Universal Robots PolyScope program: TEST_SUB_106.urp

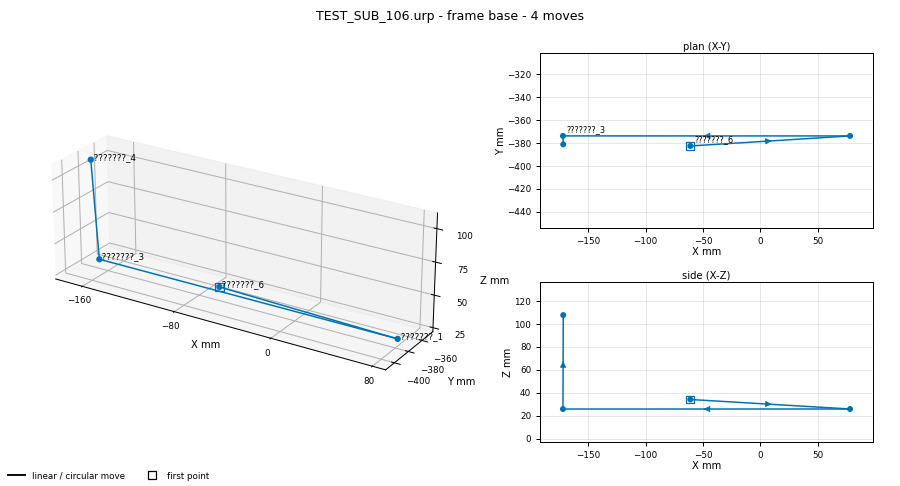
[picture p0: tool path of TEST_SUB_106.urp in frame base, 4 of 4 moves have a stored position in this frame; points joined in program order, loops and branches not executed]
Program TEST_SUB_106 (installation=GD directory=/programs/GD createdIn=5.13.0 lastSavedIn=5.13.0 robotSerialNumber=20205000017)
Calibrated DH parameters: a=[-0.000157, -0.56303, -0.236706, -0.000074, -0.000109, 0]; d=[0.181705, 47.632387, 369.599619, -417.058513, 0.119878, 0.115667]; alpha=[1.570881, -0.005074, -0.001247, 1.56886, -1.570997, 0]; deltaTheta=[0, -0.405485, 5.544791, 1.143886, -0.000009, -0.000001]
InitVariablesNode
Robot Program (runOnlyOnce=false)
  var_4 := p[0.0,0.0,0.0,CutOffPos[3],CutOffPos[4],CutOffPos[5]]
  var_5 := p[0.0,0.0,0.0,CutOffPos[3],CutOffPos[4],CutOffPos[5]]
  Script: CurrPos=get_actual_tool_flange_pose()
  CutOffPos := CurrPos
  var_1 := get_tcp_offset()
  var_2 := pose_trans(CutOffPos,var_1)
  MoveL speed 250 mm/s, acceleration 50 mm/s^2 (useActiveTCP=false) tcp=TCP_1; feature=Base
    SuppressedNode
      var_3 := get_tcp_offset()
    SuppressedNode
      Waypoint ウェイポイント_2: TCP in base x=-24.264 y=-372.872 z=25.863 mm, rx=-0.0592 ry=3.141 rz=-0.0002 rad; joints [-70.474, -66.693, -131.957, -71.332, 89.989, 17.477] deg; TCP offset x=0 y=80 z=420 mm, rx=0 ry=0 rz=0 rad
    SuppressedNode
      Wait Sleep waitTime=0.5
    Waypoint ウェイポイント_6: TCP in base x=-61.068 y=-382.464 z=34.138 mm, rx=0.7542 ry=-2.9409 rz=0.2397 rad; joints [-60.318, -53.474, -138.479, -70.758, 82.346, 0.532] deg
    Wait Sleep waitTime=0.5
  SuppressedNode
    Folder FREE_DRIVE
      Script: freedrive_mode()
      SetPayload (workpieceName=k2)
      Set NoAction tcp=ZERO
      Wait Sleep waitTime=1
      Script: end_freedrive_mode()
      Wait Condition expression=is_steady()
  SetPayload (workpieceName=k10)
  Set NoAction tcp=TCP_1
  Wait Sleep waitTime=0.5
  Folder CUTOFF_POSE
    CutOffPos := CurrPos
    var_6 := CutOffPos
    SuppressedNode
      CutOffPos := p[0.0,0.0,0.0,CutOffPos[3],CutOffPos[4],CutOffPos[5]]
    var_1 := get_tcp_offset()
    var_20 := pose_trans(pose_inv(CutOffPos),var_1)
    SuppressedNode
      CutOffPos := 
    var_4 := p[0.0,0.0,0.0,CutOffPos[3],CutOffPos[4],CutOffPos[5]]
    var_5 := p[0.0,0.0,0.0,0.0,0.0,CutOffPos[5]]
    CutOffPos := pose_trans(var_4,pose_inv(var_5))
    SuppressedNode
      CutOffPos := p[0.0,0.0,0.0,var_5[0],var_5[1],var_5[2]]
    var_20 := pose_trans(pose_inv(CutOffPos),var_1)
    var_21 := pose_trans(var_1,CutOffPos)
    var_2 := pose_trans(CutOffPos,var_1)
  Wait Condition expression=is_steady()
  SuppressedNode
    Script: CurrPos_p=get_actual_tcp_pose()
  SuppressedNode
    CircleMove (OrientationMode=UNCONSTRAINED)
  Script: set_tcp(var_2)
  SuppressedNode
    Folder TRANSFER
      Timer (action=Reset) variable(name=tm_relmove)
      Timer (action=Start) variable=tm_relmove
      ForceStartZ := CurrPos_p[2]
      Force Frame feature=Bucket; selection=[0, 0, 1, 0, 0, 0]; wrench=[0, 0, 40, 0, 0, 0]; limitsForce=[0.01, 0.01, 0.25, 0.174533, 0.174533, 0.174533]; limitsMotion=[0.1, 0.1, 0.1, 0.349066, 0.349066, 0.349066]
        Wait Condition expression=tm_relmove>GPII_TMCutOff or CurrPos_p[2]>ForceStartZ+RelMoveZ
      Timer (action=Stop) variable=tm_relmove
      If (WorkPosNo≟0)
        MoveL speed 60 mm/s, acceleration 15 mm/s^2 (useActiveTCP=false) tcp=ZERO; feature=Base
          PoseSub := pose_sub(CurrPos, pose_trans(g2GD_pos5, pose_inv(get_tcp_offset())))
          RZSub := r2d(PoseSub[5])
          If (norm(PoseSub[5])≥d2r(RZTh))
            Script: PoseSub[0]=0.0
            Script: PoseSub[1]=0.0
            Script: PoseSub[2]=0.0
            PoseAdd := pose_add(PoseSub, CurrPos)
            Waypoint Variable (Variable): variable=PoseAdd
        MoveL speed 250 mm/s, acceleration 50 mm/s^2 (useActiveTCP=false) tcp=TCP_1; feature=Base
          Waypoint Variable (Variable): variable(featureName=g2GD_pos5)
        MoveL speed 400 mm/s, acceleration 140 mm/s^2 (useActiveTCP=false) tcp=TCP_1; feature=Base
          SetPayload (workpieceName=k10)
          Waypoint Variable (Variable): variable(featureName=g2GD_pos4)
          Waypoint Variable (Variable): motionParameters(blendRadius=0.1); variable(featureName=g2GD_pos3)
          Waypoint Variable (Variable): motionParameters(jointSpeed=1.047198 jointAcceleration=1.396263 cartesianSpeed=0.4 cartesianAcceleration=0.07); variable(featureName=g2GD_pos2)
        MoveL speed 400 mm/s, acceleration 70 mm/s^2 (useActiveTCP=false) tcp=TCP_1; feature=Base
          SetPayload (workpieceName=k120)
          Waypoint Variable (Variable): motionParameters(blendRadius=0.05); variable(featureName=g2GD_pos1)
      ElseIf (WorkPosNo≟1)
        MoveL speed 60 mm/s, acceleration 15 mm/s^2 (useActiveTCP=false) tcp=ZERO; feature=Base
          PoseSub := pose_sub(CurrPos, pose_trans(g1GD_pos5, pose_inv(get_tcp_offset())))
          RZSub := r2d(PoseSub[5])
          If (norm(PoseSub[5])≥d2r(RZTh))
            Script: PoseSub[0]=0.0
            Script: PoseSub[1]=0.0
            Script: PoseSub[2]=0.0
            PoseAdd := pose_add(PoseSub, CurrPos)
            Waypoint Variable (Variable): variable=PoseAdd
        MoveL speed 250 mm/s, acceleration 50 mm/s^2 (useActiveTCP=false) tcp=TCP_1; feature=Base
          Waypoint Variable (Variable): variable(featureName=g1GD_pos5)
        MoveL speed 400 mm/s, acceleration 140 mm/s^2 (useActiveTCP=false) tcp=TCP_1; feature=Base
          SetPayload (workpieceName=k10)
          Waypoint Variable (Variable): variable(featureName=g1GD_pos3)
          Waypoint Variable (Variable): variable(featureName=g1GD_pos2)
        MoveL speed 400 mm/s, acceleration 140 mm/s^2 (useActiveTCP=false) tcp=TCP_1; feature=Base
          SetPayload (workpieceName=k120)
          Waypoint Variable (Variable): motionParameters(blendRadius=0.1); variable(featureName=g1GD_pos1)
  MoveL speed 250 mm/s, acceleration 50 mm/s^2 (useActiveTCP=true) feature=Base
    var_3 := get_tcp_offset()
    Waypoint ウェイポイント_1: TCP in base x=78.379 y=-373.699 z=25.825 mm, rx=-0.2371 ry=3.1325 rz=-0.0004 rad; joints [-56.917, -67.759, -131.362, -70.853, 89.981, 24.534] deg
    Wait Sleep waitTime=1
    Waypoint ウェイポイント_3: TCP in base x=-172.242 y=-373.664 z=25.794 mm, rx=-0.2375 ry=3.1326 rz=-0.0004 rad; joints [-88.583, -70.074, -129.994, -69.907, 89.976, -7.145] deg
    Wait Sleep waitTime=1
    Waypoint ウェイポイント_4: TCP in base x=-172.007 y=-381.075 z=107.802 mm, rx=-0.2377 ry=3.1326 rz=-0.0003 rad; joints [-88.585, -68.371, -122.486, -79.122, 89.973, -7.155] deg
    Wait Sleep waitTime=1
  Popup Message (haltProgram=false message=done! inputType=Text)
Thread スレッド_1 (runOnlyOnce=false)
  Script: CurrPos=get_actual_tool_flange_pose()
  Script: CurrPos_p=get_actual_tcp_pose()
  Script: sync()
